// TwinCAT 3 PLC project CX1D686A
// ProgramVersion: 3.1.4024.0
// libraries:
//   Tc2_Standard, * (Beckhoff Automation GmbH)
//   Tc2_System, * (Beckhoff Automation GmbH)
//   Tc3_Module, * (Beckhoff Automation GmbH)
//   VisuSymbols,3.5.10.0,System
// project tree:
//   / GlobalTextList.TcGTLO, PlcTask.TcTTO, Visualization Manager.TcVMO (not stored), VISU_TASK.TcTTO
//   GVLs/ GVL.TcGVL
//   POUs/ MAIN.TcPOU, Scale.TcPOU
//   VISUs/ Dashboard.TcVIS
// real-time tasks:
//   TASK PlcTask: cycle T#10ms, priority 20, ADS port 350
//   TASK VISU_TASK: cycle T#50000us, priority 30, ADS port 351
// I/O:
//   DEVICE Device 1 (Profinet Device CCAT (RT)), AmsNetId 5.29.104.106.2.1
//   DEVICE Device 2 (EtherCAT), AmsNetId 5.29.104.106.3.1
//     Term 1 (EK1200) [EK1200-5000 EtherCAT Power supply (2A E-Bus)]
//       Term 2 (EL1008) [EL1008 8Ch. Dig. Input 24V, 3ms]
//       Term 3 (EL2004) [EL2004 4Ch. Dig. Output 24V, 0.5A]
//       Term 4 (EL3044) [EL3044 4Ch. Ana. Input 0-20mA]
//       Term 5 (EL9011) [EL9011 End Terminal]
//   DEVICE Device 3 (EtherCAT Automation Protocol), AmsNetId 5.29.104.106.4.1
//   DEVICE Device 5 (NOV-DP-RAM)
// variable links:
//   CX1D686A/CX1D686A Instance <-> Device 1 (Profinet Device CCAT (RT))
//     PlcTask Inputs/GVL.ProfinetState <-> Inputs/DevState
//   CX1D686A/CX1D686A Instance <-> Device 2 (EtherCAT)
//     PlcTask Inputs/GVL.EtherCATState <-> Inputs/DevState
//   CX1D686A/CX1D686A Instance <-> Device 2 (EtherCAT)/Term 1 (EK1200)/Term 2 (EL1008)
//     PlcTask Inputs/GVL.DI{0..7} <-> Channel {1..8}/Input  (8 links)
//   CX1D686A/CX1D686A Instance <-> Device 2 (EtherCAT)/Term 1 (EK1200)/Term 3 (EL2004)
//     PlcTask Outputs/GVL.DO{0..3} <-> Channel {1..4}/Output  (4 links)
//   CX1D686A/CX1D686A Instance <-> Device 2 (EtherCAT)/Term 1 (EK1200)/Term 4 (EL3044)
//     PlcTask Inputs/GVL.AI{0..3} <-> AI Standard Channel {1..4}/Value  (4 links)
//   CX1D686A/CX1D686A Instance <-> Device 3 (EtherCAT Automation Protocol)
//     PlcTask Inputs/GVL.EtherCATAutoState <-> Inputs/DevState

CONFIGURATION CX1D686A
    RESOURCE PLC ON TwinCAT3
        TASK PlcTask(INTERVAL := T#10ms, PRIORITY := 20);
        TASK VISU_TASK(INTERVAL := T#40us, PRIORITY := 30);
        PROGRAM MAIN WITH PlcTask : MAIN;
        PROGRAM VisuElems_Visu_Prg WITH VISU_TASK : VisuElems.Visu_Prg;
    END_RESOURCE
END_CONFIGURATION

// ---- GVLs/GVL.TcGVL
{attribute 'qualified_only'}
VAR_GLOBAL
	// module status'
	ProfinetState AT %I* : UINT; // ProfiNet Status
	EtherCATState AT %I* : UINT; // EtherCAT Status
	EtherCATAutoState AT %I* : UINT; // EtherCAT Automation Status
	

	// digital inputs
	DI0 AT %I* : BOOL; // Green Button
	DI1 AT %I* : BOOL; // Red Button
	DI2 AT %I* : BOOL;
	DI3 AT %I* : BOOL;
	DI4 AT %I* : BOOL;
	DI5 AT %I* : BOOL;
	DI6 AT %I* : BOOL;
	DI7 AT %I* : BOOL;
	
	// digital software overrides
	DI0_OR : BOOL := FALSE; // Green Button Override
	DI1_OR : BOOL := FALSE; // Red Button Override
	
	// digital outputs
	DO0 AT %Q* : BOOL; // Green LED
	DO1 AT %Q* : BOOL; // Red LED
	DO2 AT %Q* : BOOL;
	DO3 AT %Q* : BOOL;
	
	// analog inputs
	AI0 AT %I* : INT; // 4-20mA Input 1
	AI1 AT %I* : INT; // 4-20mA Input 2
	AI2 AT %I* : INT;
	AI3 AT %I* : INT;
	
END_VAR

// ---- POUs/MAIN.TcPOU
PROGRAM MAIN
VAR
	counter : INT := 0;
	
	Setup : BOOL := TRUE;
	
	// AI Scaling to percent
	AI_Low : INT := 3375; 
	AI_High : INT := 20200;
	AI0_scaled : INT := 0;
	
	// led toggle rates (Hz)
	toggleRate : INT := 1;
	toggleRateMax : INT := 100;
	toggleRateMin : INT := 1;
	toggleEnable: BOOL := FALSE;
END_VAR

// setup
IF Setup THEN
	GVL.DO0 := FALSE;
	GVL.DO1 := TRUE;
	
	// setup finished
	Setup := FALSE;
END_IF


// main loop
counter := counter + 100;
IF counter > 30000 THEN
	counter := 0;
END_IF

// scale AI value to percent
AI0_scaled := Scale(GVL.AI0, 
					AI_High, AI_Low,
					toggleRateMax, toggleRateMin);
					
IF GVL.DI0 OR GVL.DI0_OR THEN
	toggleEnable := TRUE;
END_IF

IF GVL.DI1 OR GVL.DI1_OR THEN
	toggleEnable := FALSE;
END_IF

IF toggleEnable THEN
	IF counter > GVL.AI0 THEN
		GVL.DO0 := NOT GVL.DO0;
		GVL.DO1 := NOT GVL.DO1;
		counter := 0;
	END_IF
END_IF

END_PROGRAM

// ---- POUs/Scale.TcPOU
FUNCTION Scale : INT
VAR_INPUT
	input : INT := 0;
	in_Max : INT := 1;
	in_Min : INT := 0;
	out_Max : INT := 1;
	out_Min : INT := 0;
END_VAR
VAR
	output : INT := 0;
END_VAR


output := ((input - in_Min)/(in_Max - in_Min)*
(out_Max - out_Min)) + out_Min;

Scale := output;

END_FUNCTION

// ---- GlobalTextList.TcGTLO
TEXTLIST GlobalTextList
  808 = ''
  413 = 'AI 0'
  532 = 'AI 1'
  98 = 'OUTPUTS'
  666 = 'RUN'
  598 = 'STOP'
END_TEXTLIST

// ---- VISUs/Dashboard.TcVIS
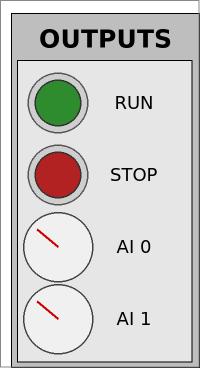
VISUALIZATION Dashboard  // 200x368
    RoundedRectangle (11,13 189x355)
    RoundedRectangle (17,60 175x302)
    Lamp1 (23,68 70x70), variable: GVL.DO0, style: Lamp-Lamp1-Green
    Lamp1 (23,140 70x70), variable: GVL.DO1, style: Lamp-Lamp1-Red
    Meter360 (23,284 70x70), value: GVL.AI1, style: Meter-Meter360-Gray, scale 0..20000
    Meter360 (23,212 70x70), value: GVL.AI1, style: Meter-Meter360-Gray, scale 0..20000
    Label (19,5 173x67), "OUTPUTS"
    Label (100,140 68x70), "STOP"
    Label (100,68 68x70), "RUN"
    Label (100,212 68x70), "AI 0"
    Label (100,284 68x70), "AI 1"
END_VISUALIZATION
